{attribute 'pack_mode' := '1'}
TYPE ST_AddPathDataIn :
STRUCT
	sCellID						: STRING(30);	// 
	iPath						: UINT;			// MM path ID (1-65536)
	bPresent					: BOOL;			// 
END_STRUCT
END_TYPE

(* stored: Version 1.1.0.1, ProductVersion 3.1.4024.5
   DUT ST_AddPathDataIn: Id {4f305d1c-bcd9-47a2-8d00-5c4bee02a267} *)
